Staubli VAL3: start.pgx

program start()
begin
  //*******************************************
  //Name: TestSoap
  //Function: test soap function
  //2012.05.28
  //y.ye@staubli.com
  //说明：这个作为一个库，被TestSoap调用
  //通过全局变量来与上位机进行交互
  //全局变量必须设定为public
  //*******************************************
end
